FUNCTION_BLOCK BlinkKoordinator (* Tamplate for a simple Basic Function Block Type *)
  (* Standard: 61499-2 *)
  (* Version 0.0, 2018-01-15, 4DIAC-IDE, 4DIAC-Consortium *)
  (* Version 1.0, 2016-05-26, AZ, fortiss GmbH *)
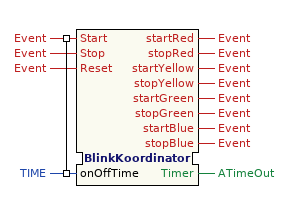
  EVENT_INPUT
    Start WITH onOffTime;
    Stop;
    Reset;
  END_EVENT
  EVENT_OUTPUT
    startRed;
    stopRed;
    startYellow;
    stopYellow;
    startGreen;
    stopGreen;
    startBlue;
    stopBlue;
  END_EVENT
  VAR_INPUT
    onOffTime : TIME;
  END_VAR
  PLUGS
    Timer : ATimeOut;
  END_PLUGS
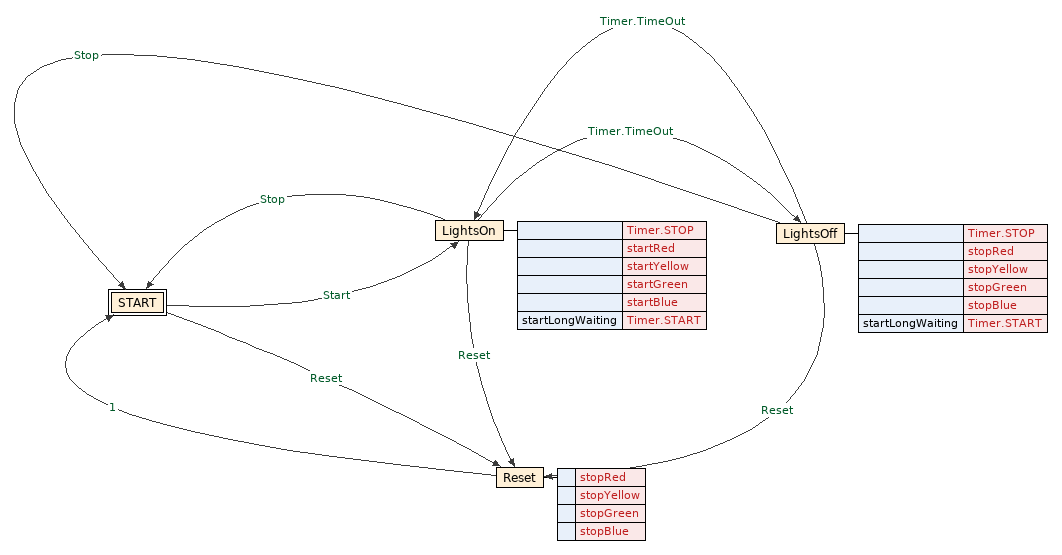
  EC_STATES
    START; (* Initial State *)
    LightsOn : -> Timer.STOP, -> startRed, -> startYellow, -> startGreen, -> startBlue, startLongWaiting -> Timer.START;
    LightsOff : -> Timer.STOP, -> stopRed, -> stopYellow, -> stopGreen, -> stopBlue, startLongWaiting -> Timer.START;
    Reset : -> stopRed, -> stopYellow, -> stopGreen, -> stopBlue;
  END_STATES
  EC_TRANSITIONS
    START TO LightsOn := Start;
    LightsOn TO LightsOff := Timer.TimeOut;
    LightsOn TO START := Stop;
    LightsOff TO START := Stop;
    LightsOff TO LightsOn := Timer.TimeOut;
    START TO Reset := Reset;
    Reset TO START := 1;
    LightsOn TO Reset := Reset;
    LightsOff TO Reset := Reset;
  END_TRANSITIONS
  ALGORITHM startLongWaiting IN ST: (* set long waiting time *)
Timer.DT := onOffTime;
  END_ALGORITHM
END_FUNCTION_BLOCK
